(* PLC project Adressering.ecp, WAGO e!COCKPIT e!COCKPIT *)
(* stored: creationDateTime 2021-01-18T14:20:23.2110188, modificationDateTime 2021-01-18T11:51:27.6823754 *)

TYPE typVAV : STRUCT
  xReady : BOOL;  (* Status adr. *)
  xEnable : BOOL;  (* Enable MP blokk *)
  xAddress : BOOL;  (* Adresserer VAV *)
  xFailed : BOOL;  (* Tilbakemelding adressering (True = SerieNr inn og ut ikke stemmer) *)
  sSetStatus : STRING;  (* Status tilbakemelding naar adresseringen er i SET step *)
  sGetStatus : STRING;  (* Status tilbakemelding naar adresseringen er i GET step *)
  iSerialNr : typSerialNo;  (* Serie NR *)
  bPort : BYTE;  (* VAV Port *)
  bAddress : BYTE;  (* VAV Address *)
  rAirVolume_SP : REAL;  (* Settpunkt 0-100% *)
  rOutPosition : REAL;  (* Vinkel *)
  rOutAirVolume_perc : REAL;  (* Luftmengde i prosent *)
  rOutAirVolume_m3h : REAL;  (* Luftmengde i m3h *)
  wSensorValue : WORD;
  rVmin : REAL;
  rVmax : REAL;  (* Max vinkel *)
  xControlRangeIncreased : BOOL;
  xMecanicalOverload : BOOL;
  xActuatorHunting : BOOL;
  xSensorError : BOOL;
  xManualOpen : BOOL;
  xManualClose : BOOL;
  vMin : REAL;  (* Min luftmengde SP / 0-100 *)
  vNorm : REAL;  (* Settpunkt ved bevegelse / 0-100 *)
  vMax : REAL;  (* Maks luftmengde SP / 0-100 *)
  vSize : REAL;  (* Max kubikk *)
  vSetpoint_m3h : REAL;  (* SP% *)
  xdontoptimize : BOOL;  (* Fjerner VAV fra Optimizer *)
END_STRUCT;
END_TYPE

{attribute 'qualified_only'}
VAR_GLOBAL  (* STLV80_360 *)
  STLV80_A_360_6D201_SQ401 : typVAV := (xEnable := TRUE, vMin := 700, vNorm := 1400, vMax := 1400, vSize := 1750, bPort := 1, bAddress := 1, iSerialNr := (wYearAndWeek := 02045, wDayAndNumber := 50010, bTypeID := 158, bTestStation := 140));  (* / *)
  STLV80_A_360_6D301_SQ501 : typVAV := (xEnable := TRUE, vMin := 3200, vNorm := 3200, vMax := 3200, vSize := 5655, bPort := 1, bAddress := 2, iSerialNr := (wYearAndWeek := 02040, wDayAndNumber := 40202, bTypeID := 158, bTestStation := 153));  (* / *)
  STLV80_A_360_6A201_SQ401 : typVAV := (xEnable := TRUE, vMin := 2025, vNorm := 4050, vMax := 4050, vSize := 5655, bPort := 1, bAddress := 3, iSerialNr := (wYearAndWeek := 02040, wDayAndNumber := 40197, bTypeID := 158, bTestStation := 140));  (* / *)
  STLV80_A_360_6A201_SQ501 : typVAV := (xEnable := TRUE, vMin := 2700, vNorm := 2700, vMax := 2700, vSize := 5655, bPort := 1, bAddress := 4, iSerialNr := (wYearAndWeek := 02040, wDayAndNumber := 40201, bTypeID := 158, bTestStation := 159));  (* / *)
  STLV80_A_360_6C206_SQ501 : typVAV := (xEnable := TRUE, vMin := 300, vNorm := 300, vMax := 300, vSize := 700, bPort := 1, bAddress := 5, iSerialNr := (wYearAndWeek := 02105, wDayAndNumber := 10009, bTypeID := 158, bTestStation := 142));  (* / *)
  STLV80_A_360_6C206_SQ401 : typVAV := (xEnable := TRUE, vMin := 375, vNorm := 750, vMax := 750, vSize := 1750, bPort := 1, bAddress := 6, iSerialNr := (wYearAndWeek := 02045, wDayAndNumber := 50010, bTypeID := 158, bTestStation := 153));  (* / *)
  STLV80_A_360_7C201_SQ401 : typVAV := (xEnable := TRUE, vMin := 200, vNorm := 200, vMax := 200, vSize := 434, bPort := 1, bAddress := 7, iSerialNr := (wYearAndWeek := 02032, wDayAndNumber := 40145, bTypeID := 158, bTestStation := 158));  (* / *)
  STLV80_A_360_7C201_SQ501 : typVAV := (xEnable := TRUE, vMin := 400, vNorm := 400, vMax := 400, vSize := 700, bPort := 1, bAddress := 8, iSerialNr := (wYearAndWeek := 02042, wDayAndNumber := 10210, bTypeID := 158, bTestStation := 153));  (* / *)
  STLV80_A_360_6G201_SQ401 : typVAV := (xEnable := TRUE, vMin := 700, vNorm := 1400, vMax := 1400, vSize := 3619, bPort := 2, bAddress := 1, iSerialNr := (wYearAndWeek := 02042, wDayAndNumber := 10209, bTypeID := 158, bTestStation := 153));  (* / *)
  STLV80_A_360_6M201_SQ503 : typVAV := (xEnable := TRUE, vMin := 850, vNorm := 850, vMax := 850, vSize := 1060, bPort := 2, bAddress := 2, iSerialNr := (wYearAndWeek := 02005, wDayAndNumber := 20125, bTypeID := 158, bTestStation := 140));  (* / *)
  STLV80_A_360_6M201_SQ403 : typVAV := (xEnable := TRUE, vMin := 1225, vNorm := 2450, vMax := 2450, vSize := 5344, bPort := 2, bAddress := 3, iSerialNr := (wYearAndWeek := 02045, wDayAndNumber := 20003, bTypeID := 158, bTestStation := 140));  (* / *)
  STLV80_A_360_6M201_SQ402 : typVAV := (xEnable := TRUE, vMin := 700, vNorm := 1400, vMax := 1400, vSize := 4524, bPort := 2, bAddress := 4, iSerialNr := (wYearAndWeek := 02042, wDayAndNumber := 10207, bTypeID := 158, bTestStation := 153));  (* / *)
  STLV80_A_360_6M201_SQ502 : typVAV := (xEnable := TRUE, vMin := 3850, vNorm := 3850, vMax := 3850, vSize := 5655, bPort := 2, bAddress := 5, iSerialNr := (wYearAndWeek := 02040, wDayAndNumber := 40196, bTypeID := 158, bTestStation := 140));  (* / *)
  STLV80_A_360_6M201_SQ501 : typVAV := (xEnable := TRUE, vMin := 2600, vNorm := 2600, vMax := 2600, vSize := 5655, bPort := 2, bAddress := 6, iSerialNr := (wYearAndWeek := 02044, wDayAndNumber := 00121, bTypeID := 158, bTestStation := 164));  (* / *)
  STLV80_A_360_6M201_SQ401 : typVAV := (xEnable := TRUE, vMin := 900, vNorm := 1800, vMax := 1800, vSize := 5344, bPort := 2, bAddress := 7, iSerialNr := (wYearAndWeek := 02045, wDayAndNumber := 20006, bTypeID := 158, bTestStation := 140));  (* / *)
  STLV80_A_360_7O201_SQ401 : typVAV := (xEnable := TRUE, vMin := 200, vNorm := 200, vMax := 200, vSize := 700, bPort := 3, bAddress := 1, iSerialNr := (wYearAndWeek := 02032, wDayAndNumber := 40155, bTypeID := 158, bTestStation := 129));  (* / *)
  STLV80_A_360_7O201_SQ501 : typVAV := (xEnable := TRUE, vMin := 400, vNorm := 400, vMax := 400, vSize := 700, bPort := 3, bAddress := 2, iSerialNr := (wYearAndWeek := 02049, wDayAndNumber := 40093, bTypeID := 158, bTestStation := 142));  (* / *)
END_VAR

FUNCTION_BLOCK fbAutAd
  VAR_INPUT
    iSerialNr : typSerialNo;
    bPort : BYTE;
    bAddress : BYTE;
    xReset : BOOL;
    xNext : BOOL;
  END_VAR
  VAR_OUTPUT
    i : INT := 0;
    xFailed : BOOL;
    sSetStatus : STRING;
    sGetStatus : STRING;
  END_VAR
  VAR
    xLearn : BOOL;
    xRetry : BOOL;
    VAV_Addressing : fbMpBusAddressing;
  END_VAR

	//Resetter forgje VAVs verdier
	IF xReset THEN
		i:= 0;
		xRetry:= FALSE;
		xFailed:= FALSE;
		sSetStatus:= '';
		sGetStatus:= '';

//Begynner paa neste VAV
	ELSIF i<1 AND xNext THEN
		VAV_Addressing
		(
			bPortMpBus:= bPort,
			bAddress:= bAddress,
			typINSerialNo:= iSerialNr,
			xLearn:= xLearn
		);
		i:= 1;

//Skriver rett port og adresse til VAV naar blokken er klar
	ELSIF VAV_Addressing.xReady AND i=1 THEN
		VAV_Addressing
		(
			xSet:= TRUE,
			xLearn:= xLearn
		);
		i:= 2;

//Spoer etter serie nr som hoerer til port og adresse
	ELSIF VAV_Addressing.xReady AND i=2 THEN
		sSetStatus:= VAV_Addressing.sStatus;
		VAV_Addressing
		(
			xGetSerialNO:= TRUE,
			xLearn:= xLearn
		);
		i:= 3;

//Sjekker om serie nr. som tilhoerer port og adressen stemmer
	ELSIF VAV_Addressing.xReady AND i=3 THEN
		sGetStatus:= VAV_Addressing.sStatus;
		//Sjekker om serie nr stemmer
		IF xRetry AND VAV_Addressing.typOUTSerialNo.wYearAndWeek <> iSerialNr.wYearAndWeek OR VAV_Addressing.typOUTSerialNo.wDayAndNumber <> iSerialNr.wDayAndNumber OR VAV_Addressing.typOUTSerialNo.bTypeID <> iSerialNr.bTypeID OR VAV_Addressing.typOUTSerialNo.bTestStation <> iSerialNr.bTestStation THEN
			xRetry:= FALSE;
			xFailed:= TRUE;
			i:=4;
		ELSIF VAV_Addressing.typOUTSerialNo.wYearAndWeek <> iSerialNr.wYearAndWeek OR VAV_Addressing.typOUTSerialNo.wDayAndNumber <> iSerialNr.wDayAndNumber OR VAV_Addressing.typOUTSerialNo.bTypeID <> iSerialNr.bTypeID OR VAV_Addressing.typOUTSerialNo.bTestStation <> iSerialNr.bTestStation THEN
			xRetry:= TRUE;
			i:=1;
		ELSE
			i:=4;
		END_IF

//Resetter xSet og xGet, og Setter Port, adresse og serie nr. og henter status
	ELSE
		VAV_Addressing
		(
			bPortMpBus:= bPort,
			bAddress:= bAddress,
			typINSerialNo:= iSerialNr,
			xLearn:= xLearn,
			xSet:= FALSE,
			xGetSerialNO:= FALSE,
			xLearn:= xLearn
		);
	END_IF
				
END_FUNCTION_BLOCK

PROGRAM PRG_VAV_Adressering
  VAR
    xReset : BOOL;
    xRun : BOOL;
    xInit : BOOL := TRUE;
    Auto : fbAutAd;
    iLinje : INT;  (* Linje som skal adresseres *)
    iVAV : INT := 1;  (* VAV(adr.) som adresseres *)
  END_VAR

					IF xReset THEN
	Auto(xReset:= TRUE);
	xInit:= TRUE;
	xReset:= FALSE;
ELSIF xRun THEN

	IF STLV80_360.STLV80_A_360_6D201_SQ401.xAddress OR (iLinje = 1 AND iVAV = 1) THEN

		IF xInit THEN
			STLV80_360.STLV80_A_360_6D201_SQ401.xEnable:= FALSE;
			Auto(
				bPort:= STLV80_360.STLV80_A_360_6D201_SQ401.bPort,
				bAddress:= STLV80_360.STLV80_A_360_6D201_SQ401.bAddress,
				iSerialNr:= STLV80_360.STLV80_A_360_6D201_SQ401.iSerialNr,
				xNext:= TRUE,
				xReset:= FALSE
				);
			xInit:= FALSE;

		ELSIF Auto.i=4 THEN
			STLV80_360.STLV80_A_360_6D201_SQ401.sSetStatus:= Auto.sSetStatus;
				STLV80_360.STLV80_A_360_6D201_SQ401.sGetStatus:= Auto.sGetStatus;
				STLV80_360.STLV80_A_360_6D201_SQ401.xFailed:= Auto.xFailed;
				STLV80_360.STLV80_A_360_6D201_SQ401.xAddress:= FALSE;
				STLV80_360.STLV80_A_360_6D201_SQ401.xEnable:= TRUE;
				xReset:= TRUE;
				iVAV:=iVAV+1;

			ELSE
				Auto(xNext:= FALSE);
			END_IF

	ELSIF STLV80_360.STLV80_A_360_6D301_SQ501.xAddress OR (iLinje = 1 AND iVAV = 2) THEN

		IF xInit THEN
			STLV80_360.STLV80_A_360_6D301_SQ501.xEnable:= FALSE;
			Auto(
				bPort:= STLV80_360.STLV80_A_360_6D301_SQ501.bPort,
				bAddress:= STLV80_360.STLV80_A_360_6D301_SQ501.bAddress,
				iSerialNr:= STLV80_360.STLV80_A_360_6D301_SQ501.iSerialNr,
				xNext:= TRUE,
				xReset:= FALSE
				);
			xInit:= FALSE;

		ELSIF Auto.i=4 THEN
			STLV80_360.STLV80_A_360_6D301_SQ501.sSetStatus:= Auto.sSetStatus;
				STLV80_360.STLV80_A_360_6D301_SQ501.sGetStatus:= Auto.sGetStatus;
				STLV80_360.STLV80_A_360_6D301_SQ501.xFailed:= Auto.xFailed;
				STLV80_360.STLV80_A_360_6D301_SQ501.xAddress:= FALSE;
				STLV80_360.STLV80_A_360_6D301_SQ501.xEnable:= TRUE;
				xReset:= TRUE;
				iVAV:=iVAV+1;

			ELSE
				Auto(xNext:= FALSE);
			END_IF

	ELSIF STLV80_360.STLV80_A_360_6A201_SQ401.xAddress OR (iLinje = 1 AND iVAV = 3) THEN

		IF xInit THEN
			STLV80_360.STLV80_A_360_6A201_SQ401.xEnable:= FALSE;
			Auto(
				bPort:= STLV80_360.STLV80_A_360_6A201_SQ401.bPort,
				bAddress:= STLV80_360.STLV80_A_360_6A201_SQ401.bAddress,
				iSerialNr:= STLV80_360.STLV80_A_360_6A201_SQ401.iSerialNr,
				xNext:= TRUE,
				xReset:= FALSE
				);
			xInit:= FALSE;

		ELSIF Auto.i=4 THEN
			STLV80_360.STLV80_A_360_6A201_SQ401.sSetStatus:= Auto.sSetStatus;
				STLV80_360.STLV80_A_360_6A201_SQ401.sGetStatus:= Auto.sGetStatus;
				STLV80_360.STLV80_A_360_6A201_SQ401.xFailed:= Auto.xFailed;
				STLV80_360.STLV80_A_360_6A201_SQ401.xAddress:= FALSE;
				STLV80_360.STLV80_A_360_6A201_SQ401.xEnable:= TRUE;
				xReset:= TRUE;
				iVAV:=iVAV+1;

			ELSE
				Auto(xNext:= FALSE);
			END_IF

	ELSIF STLV80_360.STLV80_A_360_6A201_SQ501.xAddress OR (iLinje = 1 AND iVAV = 4) THEN

		IF xInit THEN
			STLV80_360.STLV80_A_360_6A201_SQ501.xEnable:= FALSE;
			Auto(
				bPort:= STLV80_360.STLV80_A_360_6A201_SQ501.bPort,
				bAddress:= STLV80_360.STLV80_A_360_6A201_SQ501.bAddress,
				iSerialNr:= STLV80_360.STLV80_A_360_6A201_SQ501.iSerialNr,
				xNext:= TRUE,
				xReset:= FALSE
				);
			xInit:= FALSE;

		ELSIF Auto.i=4 THEN
			STLV80_360.STLV80_A_360_6A201_SQ501.sSetStatus:= Auto.sSetStatus;
				STLV80_360.STLV80_A_360_6A201_SQ501.sGetStatus:= Auto.sGetStatus;
				STLV80_360.STLV80_A_360_6A201_SQ501.xFailed:= Auto.xFailed;
				STLV80_360.STLV80_A_360_6A201_SQ501.xAddress:= FALSE;
				STLV80_360.STLV80_A_360_6A201_SQ501.xEnable:= TRUE;
				xReset:= TRUE;
				iVAV:=iVAV+1;

			ELSE
				Auto(xNext:= FALSE);
			END_IF

	ELSIF STLV80_360.STLV80_A_360_6C206_SQ501.xAddress OR (iLinje = 1 AND iVAV = 5) THEN

		IF xInit THEN
			STLV80_360.STLV80_A_360_6C206_SQ501.xEnable:= FALSE;
			Auto(
				bPort:= STLV80_360.STLV80_A_360_6C206_SQ501.bPort,
				bAddress:= STLV80_360.STLV80_A_360_6C206_SQ501.bAddress,
				iSerialNr:= STLV80_360.STLV80_A_360_6C206_SQ501.iSerialNr,
				xNext:= TRUE,
				xReset:= FALSE
				);
			xInit:= FALSE;

		ELSIF Auto.i=4 THEN
			STLV80_360.STLV80_A_360_6C206_SQ501.sSetStatus:= Auto.sSetStatus;
				STLV80_360.STLV80_A_360_6C206_SQ501.sGetStatus:= Auto.sGetStatus;
				STLV80_360.STLV80_A_360_6C206_SQ501.xFailed:= Auto.xFailed;
				STLV80_360.STLV80_A_360_6C206_SQ501.xAddress:= FALSE;
				STLV80_360.STLV80_A_360_6C206_SQ501.xEnable:= TRUE;
				xReset:= TRUE;
				iVAV:=iVAV+1;

			ELSE
				Auto(xNext:= FALSE);
			END_IF

	ELSIF STLV80_360.STLV80_A_360_6C206_SQ401.xAddress OR (iLinje = 1 AND iVAV = 6) THEN

		IF xInit THEN
			STLV80_360.STLV80_A_360_6C206_SQ401.xEnable:= FALSE;
			Auto(
				bPort:= STLV80_360.STLV80_A_360_6C206_SQ401.bPort,
				bAddress:= STLV80_360.STLV80_A_360_6C206_SQ401.bAddress,
				iSerialNr:= STLV80_360.STLV80_A_360_6C206_SQ401.iSerialNr,
				xNext:= TRUE,
				xReset:= FALSE
				);
			xInit:= FALSE;

		ELSIF Auto.i=4 THEN
			STLV80_360.STLV80_A_360_6C206_SQ401.sSetStatus:= Auto.sSetStatus;
				STLV80_360.STLV80_A_360_6C206_SQ401.sGetStatus:= Auto.sGetStatus;
				STLV80_360.STLV80_A_360_6C206_SQ401.xFailed:= Auto.xFailed;
				STLV80_360.STLV80_A_360_6C206_SQ401.xAddress:= FALSE;
				STLV80_360.STLV80_A_360_6C206_SQ401.xEnable:= TRUE;
				xReset:= TRUE;
				iVAV:=iVAV+1;

			ELSE
				Auto(xNext:= FALSE);
			END_IF

	ELSIF STLV80_360.STLV80_A_360_7C201_SQ401.xAddress OR (iLinje = 1 AND iVAV = 7) THEN

		IF xInit THEN
			STLV80_360.STLV80_A_360_7C201_SQ401.xEnable:= FALSE;
			Auto(
				bPort:= STLV80_360.STLV80_A_360_7C201_SQ401.bPort,
				bAddress:= STLV80_360.STLV80_A_360_7C201_SQ401.bAddress,
				iSerialNr:= STLV80_360.STLV80_A_360_7C201_SQ401.iSerialNr,
				xNext:= TRUE,
				xReset:= FALSE
				);
			xInit:= FALSE;

		ELSIF Auto.i=4 THEN
			STLV80_360.STLV80_A_360_7C201_SQ401.sSetStatus:= Auto.sSetStatus;
				STLV80_360.STLV80_A_360_7C201_SQ401.sGetStatus:= Auto.sGetStatus;
				STLV80_360.STLV80_A_360_7C201_SQ401.xFailed:= Auto.xFailed;
				STLV80_360.STLV80_A_360_7C201_SQ401.xAddress:= FALSE;
				STLV80_360.STLV80_A_360_7C201_SQ401.xEnable:= TRUE;
				xReset:= TRUE;
				iVAV:=iVAV+1;

			ELSE
				Auto(xNext:= FALSE);
			END_IF

	ELSIF STLV80_360.STLV80_A_360_7C201_SQ501.xAddress OR (iLinje = 1 AND iVAV = 8) THEN

		IF xInit THEN
			STLV80_360.STLV80_A_360_7C201_SQ501.xEnable:= FALSE;
			Auto(
				bPort:= STLV80_360.STLV80_A_360_7C201_SQ501.bPort,
				bAddress:= STLV80_360.STLV80_A_360_7C201_SQ501.bAddress,
				iSerialNr:= STLV80_360.STLV80_A_360_7C201_SQ501.iSerialNr,
				xNext:= TRUE,
				xReset:= FALSE
				);
			xInit:= FALSE;

		ELSIF Auto.i=4 THEN
			STLV80_360.STLV80_A_360_7C201_SQ501.sSetStatus:= Auto.sSetStatus;
				STLV80_360.STLV80_A_360_7C201_SQ501.sGetStatus:= Auto.sGetStatus;
				STLV80_360.STLV80_A_360_7C201_SQ501.xFailed:= Auto.xFailed;
				STLV80_360.STLV80_A_360_7C201_SQ501.xAddress:= FALSE;
				STLV80_360.STLV80_A_360_7C201_SQ501.xEnable:= TRUE;
				xReset:= TRUE;
				iVAV:=iVAV+1;

			ELSE
				Auto(xNext:= FALSE);
			END_IF

	ELSIF STLV80_360.STLV80_A_360_6G201_SQ401.xAddress OR (iLinje = 2 AND iVAV = 1) THEN

		IF xInit THEN
			STLV80_360.STLV80_A_360_6G201_SQ401.xEnable:= FALSE;
			Auto(
				bPort:= STLV80_360.STLV80_A_360_6G201_SQ401.bPort,
				bAddress:= STLV80_360.STLV80_A_360_6G201_SQ401.bAddress,
				iSerialNr:= STLV80_360.STLV80_A_360_6G201_SQ401.iSerialNr,
				xNext:= TRUE,
				xReset:= FALSE
				);
			xInit:= FALSE;

		ELSIF Auto.i=4 THEN
			STLV80_360.STLV80_A_360_6G201_SQ401.sSetStatus:= Auto.sSetStatus;
				STLV80_360.STLV80_A_360_6G201_SQ401.sGetStatus:= Auto.sGetStatus;
				STLV80_360.STLV80_A_360_6G201_SQ401.xFailed:= Auto.xFailed;
				STLV80_360.STLV80_A_360_6G201_SQ401.xAddress:= FALSE;
				STLV80_360.STLV80_A_360_6G201_SQ401.xEnable:= TRUE;
				xReset:= TRUE;
				iVAV:=iVAV+1;

			ELSE
				Auto(xNext:= FALSE);
			END_IF

	ELSIF STLV80_360.STLV80_A_360_6M201_SQ503.xAddress OR (iLinje = 2 AND iVAV = 2) THEN

		IF xInit THEN
			STLV80_360.STLV80_A_360_6M201_SQ503.xEnable:= FALSE;
			Auto(
				bPort:= STLV80_360.STLV80_A_360_6M201_SQ503.bPort,
				bAddress:= STLV80_360.STLV80_A_360_6M201_SQ503.bAddress,
				iSerialNr:= STLV80_360.STLV80_A_360_6M201_SQ503.iSerialNr,
				xNext:= TRUE,
				xReset:= FALSE
				);
			xInit:= FALSE;

		ELSIF Auto.i=4 THEN
			STLV80_360.STLV80_A_360_6M201_SQ503.sSetStatus:= Auto.sSetStatus;
				STLV80_360.STLV80_A_360_6M201_SQ503.sGetStatus:= Auto.sGetStatus;
				STLV80_360.STLV80_A_360_6M201_SQ503.xFailed:= Auto.xFailed;
				STLV80_360.STLV80_A_360_6M201_SQ503.xAddress:= FALSE;
				STLV80_360.STLV80_A_360_6M201_SQ503.xEnable:= TRUE;
				xReset:= TRUE;
				iVAV:=iVAV+1;

			ELSE
				Auto(xNext:= FALSE);
			END_IF

	ELSIF STLV80_360.STLV80_A_360_6M201_SQ403.xAddress OR (iLinje = 2 AND iVAV = 3) THEN

		IF xInit THEN
			STLV80_360.STLV80_A_360_6M201_SQ403.xEnable:= FALSE;
			Auto(
				bPort:= STLV80_360.STLV80_A_360_6M201_SQ403.bPort,
				bAddress:= STLV80_360.STLV80_A_360_6M201_SQ403.bAddress,
				iSerialNr:= STLV80_360.STLV80_A_360_6M201_SQ403.iSerialNr,
				xNext:= TRUE,
				xReset:= FALSE
				);
			xInit:= FALSE;

		ELSIF Auto.i=4 THEN
			STLV80_360.STLV80_A_360_6M201_SQ403.sSetStatus:= Auto.sSetStatus;
				STLV80_360.STLV80_A_360_6M201_SQ403.sGetStatus:= Auto.sGetStatus;
				STLV80_360.STLV80_A_360_6M201_SQ403.xFailed:= Auto.xFailed;
				STLV80_360.STLV80_A_360_6M201_SQ403.xAddress:= FALSE;
				STLV80_360.STLV80_A_360_6M201_SQ403.xEnable:= TRUE;
				xReset:= TRUE;
				iVAV:=iVAV+1;

			ELSE
				Auto(xNext:= FALSE);
			END_IF

	ELSIF STLV80_360.STLV80_A_360_6M201_SQ402.xAddress OR (iLinje = 2 AND iVAV = 4) THEN

		IF xInit THEN
			STLV80_360.STLV80_A_360_6M201_SQ402.xEnable:= FALSE;
			Auto(
				bPort:= STLV80_360.STLV80_A_360_6M201_SQ402.bPort,
				bAddress:= STLV80_360.STLV80_A_360_6M201_SQ402.bAddress,
				iSerialNr:= STLV80_360.STLV80_A_360_6M201_SQ402.iSerialNr,
				xNext:= TRUE,
				xReset:= FALSE
				);
			xInit:= FALSE;

		ELSIF Auto.i=4 THEN
			STLV80_360.STLV80_A_360_6M201_SQ402.sSetStatus:= Auto.sSetStatus;
				STLV80_360.STLV80_A_360_6M201_SQ402.sGetStatus:= Auto.sGetStatus;
				STLV80_360.STLV80_A_360_6M201_SQ402.xFailed:= Auto.xFailed;
				STLV80_360.STLV80_A_360_6M201_SQ402.xAddress:= FALSE;
				STLV80_360.STLV80_A_360_6M201_SQ402.xEnable:= TRUE;
				xReset:= TRUE;
				iVAV:=iVAV+1;

			ELSE
				Auto(xNext:= FALSE);
			END_IF

	ELSIF STLV80_360.STLV80_A_360_6M201_SQ502.xAddress OR (iLinje = 2 AND iVAV = 5) THEN

		IF xInit THEN
			STLV80_360.STLV80_A_360_6M201_SQ502.xEnable:= FALSE;
			Auto(
				bPort:= STLV80_360.STLV80_A_360_6M201_SQ502.bPort,
				bAddress:= STLV80_360.STLV80_A_360_6M201_SQ502.bAddress,
				iSerialNr:= STLV80_360.STLV80_A_360_6M201_SQ502.iSerialNr,
				xNext:= TRUE,
				xReset:= FALSE
				);
			xInit:= FALSE;

		ELSIF Auto.i=4 THEN
			STLV80_360.STLV80_A_360_6M201_SQ502.sSetStatus:= Auto.sSetStatus;
				STLV80_360.STLV80_A_360_6M201_SQ502.sGetStatus:= Auto.sGetStatus;
				STLV80_360.STLV80_A_360_6M201_SQ502.xFailed:= Auto.xFailed;
				STLV80_360.STLV80_A_360_6M201_SQ502.xAddress:= FALSE;
				STLV80_360.STLV80_A_360_6M201_SQ502.xEnable:= TRUE;
				xReset:= TRUE;
				iVAV:=iVAV+1;

			ELSE
				Auto(xNext:= FALSE);
			END_IF

	ELSIF STLV80_360.STLV80_A_360_6M201_SQ501.xAddress OR (iLinje = 2 AND iVAV = 6) THEN

		IF xInit THEN
			STLV80_360.STLV80_A_360_6M201_SQ501.xEnable:= FALSE;
			Auto(
				bPort:= STLV80_360.STLV80_A_360_6M201_SQ501.bPort,
				bAddress:= STLV80_360.STLV80_A_360_6M201_SQ501.bAddress,
				iSerialNr:= STLV80_360.STLV80_A_360_6M201_SQ501.iSerialNr,
				xNext:= TRUE,
				xReset:= FALSE
				);
			xInit:= FALSE;

		ELSIF Auto.i=4 THEN
			STLV80_360.STLV80_A_360_6M201_SQ501.sSetStatus:= Auto.sSetStatus;
				STLV80_360.STLV80_A_360_6M201_SQ501.sGetStatus:= Auto.sGetStatus;
				STLV80_360.STLV80_A_360_6M201_SQ501.xFailed:= Auto.xFailed;
				STLV80_360.STLV80_A_360_6M201_SQ501.xAddress:= FALSE;
				STLV80_360.STLV80_A_360_6M201_SQ501.xEnable:= TRUE;
				xReset:= TRUE;
				iVAV:=iVAV+1;

			ELSE
				Auto(xNext:= FALSE);
			END_IF

	ELSIF STLV80_360.STLV80_A_360_6M201_SQ401.xAddress OR (iLinje = 2 AND iVAV = 7) THEN

		IF xInit THEN
			STLV80_360.STLV80_A_360_6M201_SQ401.xEnable:= FALSE;
			Auto(
				bPort:= STLV80_360.STLV80_A_360_6M201_SQ401.bPort,
				bAddress:= STLV80_360.STLV80_A_360_6M201_SQ401.bAddress,
				iSerialNr:= STLV80_360.STLV80_A_360_6M201_SQ401.iSerialNr,
				xNext:= TRUE,
				xReset:= FALSE
				);
			xInit:= FALSE;

		ELSIF Auto.i=4 THEN
			STLV80_360.STLV80_A_360_6M201_SQ401.sSetStatus:= Auto.sSetStatus;
				STLV80_360.STLV80_A_360_6M201_SQ401.sGetStatus:= Auto.sGetStatus;
				STLV80_360.STLV80_A_360_6M201_SQ401.xFailed:= Auto.xFailed;
				STLV80_360.STLV80_A_360_6M201_SQ401.xAddress:= FALSE;
				STLV80_360.STLV80_A_360_6M201_SQ401.xEnable:= TRUE;
				xReset:= TRUE;
				iVAV:=iVAV+1;

			ELSE
				Auto(xNext:= FALSE);
			END_IF

	ELSIF STLV80_360.STLV80_A_360_7O201_SQ401.xAddress OR (iLinje = 3 AND iVAV = 1) THEN

		IF xInit THEN
			STLV80_360.STLV80_A_360_7O201_SQ401.xEnable:= FALSE;
			Auto(
				bPort:= STLV80_360.STLV80_A_360_7O201_SQ401.bPort,
				bAddress:= STLV80_360.STLV80_A_360_7O201_SQ401.bAddress,
				iSerialNr:= STLV80_360.STLV80_A_360_7O201_SQ401.iSerialNr,
				xNext:= TRUE,
				xReset:= FALSE
				);
			xInit:= FALSE;

		ELSIF Auto.i=4 THEN
			STLV80_360.STLV80_A_360_7O201_SQ401.sSetStatus:= Auto.sSetStatus;
				STLV80_360.STLV80_A_360_7O201_SQ401.sGetStatus:= Auto.sGetStatus;
				STLV80_360.STLV80_A_360_7O201_SQ401.xFailed:= Auto.xFailed;
				STLV80_360.STLV80_A_360_7O201_SQ401.xAddress:= FALSE;
				STLV80_360.STLV80_A_360_7O201_SQ401.xEnable:= TRUE;
				xReset:= TRUE;
				iVAV:=iVAV+1;

			ELSE
				Auto(xNext:= FALSE);
			END_IF

	ELSIF STLV80_360.STLV80_A_360_7O201_SQ501.xAddress OR (iLinje = 3 AND iVAV = 2) THEN

		IF xInit THEN
			STLV80_360.STLV80_A_360_7O201_SQ501.xEnable:= FALSE;
			Auto(
				bPort:= STLV80_360.STLV80_A_360_7O201_SQ501.bPort,
				bAddress:= STLV80_360.STLV80_A_360_7O201_SQ501.bAddress,
				iSerialNr:= STLV80_360.STLV80_A_360_7O201_SQ501.iSerialNr,
				xNext:= TRUE,
				xReset:= FALSE
				);
			xInit:= FALSE;

		ELSIF Auto.i=4 THEN
			STLV80_360.STLV80_A_360_7O201_SQ501.sSetStatus:= Auto.sSetStatus;
				STLV80_360.STLV80_A_360_7O201_SQ501.sGetStatus:= Auto.sGetStatus;
				STLV80_360.STLV80_A_360_7O201_SQ501.xFailed:= Auto.xFailed;
				STLV80_360.STLV80_A_360_7O201_SQ501.xAddress:= FALSE;
				STLV80_360.STLV80_A_360_7O201_SQ501.xEnable:= TRUE;
				xReset:= TRUE;
				iVAV:=iVAV+1;

			ELSE
				Auto(xNext:= FALSE);
			END_IF

	ELSIF iVAV > 8 THEN
			iVAV:= 0;
		ELSIF iVAV > 0  THEN
			iVAV:= (iVAV+1);
		END_IF
END_IF

				
END_PROGRAM

PROGRAM PRG_MP1
  VAR
    xSet : BOOL;  (* Felles *)
    xRead : BOOL;
    FbMpbusMaster_1 : FbMpbusMaster;  (* Master *)
    oStatus_M1 : WagoSysErrorBase.FbResult;
    sStatus_M1 : STRING;
    FbMpbus_1 : FbMpBusVav;  (* Linje 1. Adresse 1. VAV STLV80_A_360_6D201_SQ401 *)
    oStatus_1 : WagoSysErrorBase.FbResult;
    sStatus_1 : STRING;
    FbMpbus_2 : FbMpBusVav;  (* Linje 1. Adresse 2. VAV STLV80_A_360_6D301_SQ501 *)
    oStatus_2 : WagoSysErrorBase.FbResult;
    sStatus_2 : STRING;
    FbMpbus_3 : FbMpBusVav;  (* Linje 1. Adresse 3. VAV STLV80_A_360_6A201_SQ401 *)
    oStatus_3 : WagoSysErrorBase.FbResult;
    sStatus_3 : STRING;
    FbMpbus_4 : FbMpBusVav;  (* Linje 1. Adresse 4. VAV STLV80_A_360_6A201_SQ501 *)
    oStatus_4 : WagoSysErrorBase.FbResult;
    sStatus_4 : STRING;
    FbMpbus_5 : FbMpBusVav;  (* Linje 1. Adresse 5. VAV STLV80_A_360_6C206_SQ501 *)
    oStatus_5 : WagoSysErrorBase.FbResult;
    sStatus_5 : STRING;
    FbMpbus_6 : FbMpBusVav;  (* Linje 1. Adresse 6. VAV STLV80_A_360_6C206_SQ401 *)
    oStatus_6 : WagoSysErrorBase.FbResult;
    sStatus_6 : STRING;
    FbMpbus_7 : FbMpBusVav;  (* Linje 1. Adresse 7. VAV STLV80_A_360_7C201_SQ401 *)
    oStatus_7 : WagoSysErrorBase.FbResult;
    sStatus_7 : STRING;
    FbMpbus_8 : FbMpBusVav;  (* Linje 1. Adresse 8. VAV STLV80_A_360_7C201_SQ501 *)
    oStatus_8 : WagoSysErrorBase.FbResult;
    sStatus_8 : STRING;
  END_VAR

(* CFC diagram, written out as Structured Text *)
FbMpbusMaster_1(I_Port := IoConfig_Globals.MP_Bus_Master, bPortMpBus := 1);
oStatus_M1 := FbMpbusMaster_1.oStatus;
sStatus_M1 := FbMpbusMaster_1.sStatus;
(* STLV80_A_360_6D201_SQ401 *)
FbMpbus_1(xEnable := STLV80_360.STLV80_A_360_6D201_SQ401.xEnable, bPortMpBus := 1, bAddress := 1, tCycleTime := t#500ms, rAirVolume := STLV80_360.STLV80_A_360_6D201_SQ401.rAirVolume_SP, rMinAirVolume := 0, rMaxAirVolume := 100, xSet := xSet, xRead := xRead, bSensorType := 0, xManualOpen := STLV80_360.STLV80_A_360_6D201_SQ401.xManualOpen, xManualClose := STLV80_360.STLV80_A_360_6D201_SQ401.xManualClose);
oStatus_1 := FbMpbus_1.oStatus;
sStatus_1 := FbMpbus_1.sStatus;
STLV80_360.STLV80_A_360_6D201_SQ401.xReady := FbMpbus_1.xReady;
STLV80_360.STLV80_A_360_6D201_SQ401.rOutPosition := FbMpbus_1.rOutPosition;
STLV80_360.STLV80_A_360_6D201_SQ401.rOutAirVolume_perc := FbMpbus_1.rOutAirVolume_perc;
STLV80_360.STLV80_A_360_6D201_SQ401.rOutAirVolume_m3h := FbMpbus_1.rOutAirVolume_m3_h;
STLV80_360.STLV80_A_360_6D201_SQ401.wSensorValue := FbMpbus_1.wSensorValue;
STLV80_360.STLV80_A_360_6D201_SQ401.rVmin := FbMpbus_1.rVmin;
STLV80_360.STLV80_A_360_6D201_SQ401.rVmax := FbMpbus_1.rVmax;
STLV80_360.STLV80_A_360_6D201_SQ401.xControlRangeIncreased := FbMpbus_1.xControlRangeIncreased;
STLV80_360.STLV80_A_360_6D201_SQ401.xMecanicalOverload := FbMpbus_1.xMecanicalOverload;
STLV80_360.STLV80_A_360_6D201_SQ401.xActuatorHunting := FbMpbus_1.xActuatorHunting;
STLV80_360.STLV80_A_360_6D201_SQ401.xSensorError := FbMpbus_1.xSensorError;
(* STLV80_A_360_6D301_SQ501 *)
FbMpbus_2(xEnable := STLV80_360.STLV80_A_360_6D301_SQ501.xEnable, bPortMpBus := 1, bAddress := 2, tCycleTime := t#500ms, rAirVolume := STLV80_360.STLV80_A_360_6D301_SQ501.rAirVolume_SP, rMinAirVolume := 0, rMaxAirVolume := 100, xSet := xSet, xRead := xRead, bSensorType := 0, xManualOpen := STLV80_360.STLV80_A_360_6D301_SQ501.xManualOpen, xManualClose := STLV80_360.STLV80_A_360_6D301_SQ501.xManualClose);
oStatus_2 := FbMpbus_2.oStatus;
sStatus_2 := FbMpbus_2.sStatus;
STLV80_360.STLV80_A_360_6D301_SQ501.xReady := FbMpbus_2.xReady;
STLV80_360.STLV80_A_360_6D301_SQ501.rOutPosition := FbMpbus_2.rOutPosition;
STLV80_360.STLV80_A_360_6D301_SQ501.rOutAirVolume_perc := FbMpbus_2.rOutAirVolume_perc;
STLV80_360.STLV80_A_360_6D301_SQ501.rOutAirVolume_m3h := FbMpbus_2.rOutAirVolume_m3_h;
STLV80_360.STLV80_A_360_6D301_SQ501.wSensorValue := FbMpbus_2.wSensorValue;
STLV80_360.STLV80_A_360_6D301_SQ501.rVmin := FbMpbus_2.rVmin;
STLV80_360.STLV80_A_360_6D301_SQ501.rVmax := FbMpbus_2.rVmax;
STLV80_360.STLV80_A_360_6D301_SQ501.xControlRangeIncreased := FbMpbus_2.xControlRangeIncreased;
STLV80_360.STLV80_A_360_6D301_SQ501.xMecanicalOverload := FbMpbus_2.xMecanicalOverload;
STLV80_360.STLV80_A_360_6D301_SQ501.xActuatorHunting := FbMpbus_2.xActuatorHunting;
STLV80_360.STLV80_A_360_6D301_SQ501.xSensorError := FbMpbus_2.xSensorError;
(* STLV80_A_360_6A201_SQ401 *)
FbMpbus_3(xEnable := STLV80_360.STLV80_A_360_6A201_SQ401.xEnable, bPortMpBus := 1, bAddress := 3, tCycleTime := t#500ms, rAirVolume := STLV80_360.STLV80_A_360_6A201_SQ401.rAirVolume_SP, rMinAirVolume := 0, rMaxAirVolume := 100, xSet := xSet, xRead := xRead, bSensorType := 0, xManualOpen := STLV80_360.STLV80_A_360_6A201_SQ401.xManualOpen, xManualClose := STLV80_360.STLV80_A_360_6A201_SQ401.xManualClose);
oStatus_3 := FbMpbus_3.oStatus;
sStatus_3 := FbMpbus_3.sStatus;
STLV80_360.STLV80_A_360_6A201_SQ401.xReady := FbMpbus_3.xReady;
STLV80_360.STLV80_A_360_6A201_SQ401.rOutPosition := FbMpbus_3.rOutPosition;
STLV80_360.STLV80_A_360_6A201_SQ401.rOutAirVolume_perc := FbMpbus_3.rOutAirVolume_perc;
STLV80_360.STLV80_A_360_6A201_SQ401.rOutAirVolume_m3h := FbMpbus_3.rOutAirVolume_m3_h;
STLV80_360.STLV80_A_360_6A201_SQ401.wSensorValue := FbMpbus_3.wSensorValue;
STLV80_360.STLV80_A_360_6A201_SQ401.rVmin := FbMpbus_3.rVmin;
STLV80_360.STLV80_A_360_6A201_SQ401.rVmax := FbMpbus_3.rVmax;
STLV80_360.STLV80_A_360_6A201_SQ401.xControlRangeIncreased := FbMpbus_3.xControlRangeIncreased;
STLV80_360.STLV80_A_360_6A201_SQ401.xMecanicalOverload := FbMpbus_3.xMecanicalOverload;
STLV80_360.STLV80_A_360_6A201_SQ401.xActuatorHunting := FbMpbus_3.xActuatorHunting;
STLV80_360.STLV80_A_360_6A201_SQ401.xSensorError := FbMpbus_3.xSensorError;
(* STLV80_A_360_6A201_SQ501 *)
FbMpbus_4(xEnable := STLV80_360.STLV80_A_360_6A201_SQ501.xEnable, bPortMpBus := 1, bAddress := 4, tCycleTime := t#500ms, rAirVolume := STLV80_360.STLV80_A_360_6A201_SQ501.rAirVolume_SP, rMinAirVolume := 0, rMaxAirVolume := 100, xSet := xSet, xRead := xRead, bSensorType := 0, xManualOpen := STLV80_360.STLV80_A_360_6A201_SQ501.xManualOpen, xManualClose := STLV80_360.STLV80_A_360_6A201_SQ501.xManualClose);
oStatus_4 := FbMpbus_4.oStatus;
sStatus_4 := FbMpbus_4.sStatus;
STLV80_360.STLV80_A_360_6A201_SQ501.xReady := FbMpbus_4.xReady;
STLV80_360.STLV80_A_360_6A201_SQ501.rOutPosition := FbMpbus_4.rOutPosition;
STLV80_360.STLV80_A_360_6A201_SQ501.rOutAirVolume_perc := FbMpbus_4.rOutAirVolume_perc;
STLV80_360.STLV80_A_360_6A201_SQ501.rOutAirVolume_m3h := FbMpbus_4.rOutAirVolume_m3_h;
STLV80_360.STLV80_A_360_6A201_SQ501.wSensorValue := FbMpbus_4.wSensorValue;
STLV80_360.STLV80_A_360_6A201_SQ501.rVmin := FbMpbus_4.rVmin;
STLV80_360.STLV80_A_360_6A201_SQ501.rVmax := FbMpbus_4.rVmax;
STLV80_360.STLV80_A_360_6A201_SQ501.xControlRangeIncreased := FbMpbus_4.xControlRangeIncreased;
STLV80_360.STLV80_A_360_6A201_SQ501.xMecanicalOverload := FbMpbus_4.xMecanicalOverload;
STLV80_360.STLV80_A_360_6A201_SQ501.xActuatorHunting := FbMpbus_4.xActuatorHunting;
STLV80_360.STLV80_A_360_6A201_SQ501.xSensorError := FbMpbus_4.xSensorError;
(* STLV80_A_360_6C206_SQ501 *)
FbMpbus_5(xEnable := STLV80_360.STLV80_A_360_6C206_SQ501.xEnable, bPortMpBus := 1, bAddress := 5, tCycleTime := t#500ms, rAirVolume := STLV80_360.STLV80_A_360_6C206_SQ501.rAirVolume_SP, rMinAirVolume := 0, rMaxAirVolume := 100, xSet := xSet, xRead := xRead, bSensorType := 0, xManualOpen := STLV80_360.STLV80_A_360_6C206_SQ501.xManualOpen, xManualClose := STLV80_360.STLV80_A_360_6C206_SQ501.xManualClose);
oStatus_5 := FbMpbus_5.oStatus;
sStatus_5 := FbMpbus_5.sStatus;
STLV80_360.STLV80_A_360_6C206_SQ501.xReady := FbMpbus_5.xReady;
STLV80_360.STLV80_A_360_6C206_SQ501.rOutPosition := FbMpbus_5.rOutPosition;
STLV80_360.STLV80_A_360_6C206_SQ501.rOutAirVolume_perc := FbMpbus_5.rOutAirVolume_perc;
STLV80_360.STLV80_A_360_6C206_SQ501.rOutAirVolume_m3h := FbMpbus_5.rOutAirVolume_m3_h;
STLV80_360.STLV80_A_360_6C206_SQ501.wSensorValue := FbMpbus_5.wSensorValue;
STLV80_360.STLV80_A_360_6C206_SQ501.rVmin := FbMpbus_5.rVmin;
STLV80_360.STLV80_A_360_6C206_SQ501.rVmax := FbMpbus_5.rVmax;
STLV80_360.STLV80_A_360_6C206_SQ501.xControlRangeIncreased := FbMpbus_5.xControlRangeIncreased;
STLV80_360.STLV80_A_360_6C206_SQ501.xMecanicalOverload := FbMpbus_5.xMecanicalOverload;
STLV80_360.STLV80_A_360_6C206_SQ501.xActuatorHunting := FbMpbus_5.xActuatorHunting;
STLV80_360.STLV80_A_360_6C206_SQ501.xSensorError := FbMpbus_5.xSensorError;
(* STLV80_A_360_6C206_SQ401 *)
FbMpbus_6(xEnable := STLV80_360.STLV80_A_360_6C206_SQ401.xEnable, bPortMpBus := 1, bAddress := 6, tCycleTime := t#500ms, rAirVolume := STLV80_360.STLV80_A_360_6C206_SQ401.rAirVolume_SP, rMinAirVolume := 0, rMaxAirVolume := 100, xSet := xSet, xRead := xRead, bSensorType := 0, xManualOpen := STLV80_360.STLV80_A_360_6C206_SQ401.xManualOpen, xManualClose := STLV80_360.STLV80_A_360_6C206_SQ401.xManualClose);
oStatus_6 := FbMpbus_6.oStatus;
sStatus_6 := FbMpbus_6.sStatus;
STLV80_360.STLV80_A_360_6C206_SQ401.xReady := FbMpbus_6.xReady;
STLV80_360.STLV80_A_360_6C206_SQ401.rOutPosition := FbMpbus_6.rOutPosition;
STLV80_360.STLV80_A_360_6C206_SQ401.rOutAirVolume_perc := FbMpbus_6.rOutAirVolume_perc;
STLV80_360.STLV80_A_360_6C206_SQ401.rOutAirVolume_m3h := FbMpbus_6.rOutAirVolume_m3_h;
STLV80_360.STLV80_A_360_6C206_SQ401.wSensorValue := FbMpbus_6.wSensorValue;
STLV80_360.STLV80_A_360_6C206_SQ401.rVmin := FbMpbus_6.rVmin;
STLV80_360.STLV80_A_360_6C206_SQ401.rVmax := FbMpbus_6.rVmax;
STLV80_360.STLV80_A_360_6C206_SQ401.xControlRangeIncreased := FbMpbus_6.xControlRangeIncreased;
STLV80_360.STLV80_A_360_6C206_SQ401.xMecanicalOverload := FbMpbus_6.xMecanicalOverload;
STLV80_360.STLV80_A_360_6C206_SQ401.xActuatorHunting := FbMpbus_6.xActuatorHunting;
STLV80_360.STLV80_A_360_6C206_SQ401.xSensorError := FbMpbus_6.xSensorError;
(* STLV80_A_360_7C201_SQ401 *)
FbMpbus_7(xEnable := STLV80_360.STLV80_A_360_7C201_SQ401.xEnable, bPortMpBus := 1, bAddress := 7, tCycleTime := t#500ms, rAirVolume := STLV80_360.STLV80_A_360_7C201_SQ401.rAirVolume_SP, rMinAirVolume := 0, rMaxAirVolume := 100, xSet := xSet, xRead := xRead, bSensorType := 0, xManualOpen := STLV80_360.STLV80_A_360_7C201_SQ401.xManualOpen, xManualClose := STLV80_360.STLV80_A_360_7C201_SQ401.xManualClose);
oStatus_7 := FbMpbus_7.oStatus;
sStatus_7 := FbMpbus_7.sStatus;
STLV80_360.STLV80_A_360_7C201_SQ401.xReady := FbMpbus_7.xReady;
STLV80_360.STLV80_A_360_7C201_SQ401.rOutPosition := FbMpbus_7.rOutPosition;
STLV80_360.STLV80_A_360_7C201_SQ401.rOutAirVolume_perc := FbMpbus_7.rOutAirVolume_perc;
STLV80_360.STLV80_A_360_7C201_SQ401.rOutAirVolume_m3h := FbMpbus_7.rOutAirVolume_m3_h;
STLV80_360.STLV80_A_360_7C201_SQ401.wSensorValue := FbMpbus_7.wSensorValue;
STLV80_360.STLV80_A_360_7C201_SQ401.rVmin := FbMpbus_7.rVmin;
STLV80_360.STLV80_A_360_7C201_SQ401.rVmax := FbMpbus_7.rVmax;
STLV80_360.STLV80_A_360_7C201_SQ401.xControlRangeIncreased := FbMpbus_7.xControlRangeIncreased;
STLV80_360.STLV80_A_360_7C201_SQ401.xMecanicalOverload := FbMpbus_7.xMecanicalOverload;
STLV80_360.STLV80_A_360_7C201_SQ401.xActuatorHunting := FbMpbus_7.xActuatorHunting;
STLV80_360.STLV80_A_360_7C201_SQ401.xSensorError := FbMpbus_7.xSensorError;
(* STLV80_A_360_7C201_SQ501 *)
FbMpbus_8(xEnable := STLV80_360.STLV80_A_360_7C201_SQ501.xEnable, bPortMpBus := 1, bAddress := 8, tCycleTime := t#500ms, rAirVolume := STLV80_360.STLV80_A_360_7C201_SQ501.rAirVolume_SP, rMinAirVolume := 0, rMaxAirVolume := 100, xSet := xSet, xRead := xRead, bSensorType := 0, xManualOpen := STLV80_360.STLV80_A_360_7C201_SQ501.xManualOpen, xManualClose := STLV80_360.STLV80_A_360_7C201_SQ501.xManualClose);
oStatus_8 := FbMpbus_8.oStatus;
sStatus_8 := FbMpbus_8.sStatus;
STLV80_360.STLV80_A_360_7C201_SQ501.xReady := FbMpbus_8.xReady;
STLV80_360.STLV80_A_360_7C201_SQ501.rOutPosition := FbMpbus_8.rOutPosition;
STLV80_360.STLV80_A_360_7C201_SQ501.rOutAirVolume_perc := FbMpbus_8.rOutAirVolume_perc;
STLV80_360.STLV80_A_360_7C201_SQ501.rOutAirVolume_m3h := FbMpbus_8.rOutAirVolume_m3_h;
STLV80_360.STLV80_A_360_7C201_SQ501.wSensorValue := FbMpbus_8.wSensorValue;
STLV80_360.STLV80_A_360_7C201_SQ501.rVmin := FbMpbus_8.rVmin;
STLV80_360.STLV80_A_360_7C201_SQ501.rVmax := FbMpbus_8.rVmax;
STLV80_360.STLV80_A_360_7C201_SQ501.xControlRangeIncreased := FbMpbus_8.xControlRangeIncreased;
STLV80_360.STLV80_A_360_7C201_SQ501.xMecanicalOverload := FbMpbus_8.xMecanicalOverload;
STLV80_360.STLV80_A_360_7C201_SQ501.xActuatorHunting := FbMpbus_8.xActuatorHunting;
STLV80_360.STLV80_A_360_7C201_SQ501.xSensorError := FbMpbus_8.xSensorError;
END_PROGRAM

PROGRAM PRG_MP2
  VAR
    xSet : BOOL;  (* Felles *)
    xRead : BOOL;
    FbMpbusMaster_2 : FbMpbusMaster;  (* Master *)
    oStatus_M2 : WagoSysErrorBase.FbResult;
    sStatus_M2 : STRING;
    FbMpbus_1 : FbMpBusVav;  (* Linje 2. Adresse 1. VAV STLV80_A_360_6G201_SQ401 *)
    oStatus_1 : WagoSysErrorBase.FbResult;
    sStatus_1 : STRING;
    FbMpbus_2 : FbMpBusVav;  (* Linje 2. Adresse 2. VAV STLV80_A_360_6M201_SQ503 *)
    oStatus_2 : WagoSysErrorBase.FbResult;
    sStatus_2 : STRING;
    FbMpbus_3 : FbMpBusVav;  (* Linje 2. Adresse 3. VAV STLV80_A_360_6M201_SQ403 *)
    oStatus_3 : WagoSysErrorBase.FbResult;
    sStatus_3 : STRING;
    FbMpbus_4 : FbMpBusVav;  (* Linje 2. Adresse 4. VAV STLV80_A_360_6M201_SQ402 *)
    oStatus_4 : WagoSysErrorBase.FbResult;
    sStatus_4 : STRING;
    FbMpbus_5 : FbMpBusVav;  (* Linje 2. Adresse 5. VAV STLV80_A_360_6M201_SQ502 *)
    oStatus_5 : WagoSysErrorBase.FbResult;
    sStatus_5 : STRING;
    FbMpbus_6 : FbMpBusVav;  (* Linje 2. Adresse 6. VAV STLV80_A_360_6M201_SQ501 *)
    oStatus_6 : WagoSysErrorBase.FbResult;
    sStatus_6 : STRING;
    FbMpbus_7 : FbMpBusVav;  (* Linje 2. Adresse 7. VAV STLV80_A_360_6M201_SQ401 *)
    oStatus_7 : WagoSysErrorBase.FbResult;
    sStatus_7 : STRING;
  END_VAR

(* CFC diagram, written out as Structured Text *)
FbMpbusMaster_2(I_Port := IoConfig_Globals.MP_Bus_Master_1, bPortMpBus := 2);
oStatus_M2 := FbMpbusMaster_2.oStatus;
sStatus_M2 := FbMpbusMaster_2.sStatus;
(* STLV80_A_360_6G201_SQ401 *)
FbMpbus_1(xEnable := STLV80_360.STLV80_A_360_6G201_SQ401.xEnable, bPortMpBus := 2, bAddress := 1, tCycleTime := t#500ms, rAirVolume := STLV80_360.STLV80_A_360_6G201_SQ401.rAirVolume_SP, rMinAirVolume := 0, rMaxAirVolume := 100, xSet := xSet, xRead := xRead, bSensorType := 0, xManualOpen := STLV80_360.STLV80_A_360_6G201_SQ401.xManualOpen, xManualClose := STLV80_360.STLV80_A_360_6G201_SQ401.xManualClose);
oStatus_1 := FbMpbus_1.oStatus;
sStatus_1 := FbMpbus_1.sStatus;
STLV80_360.STLV80_A_360_6G201_SQ401.xReady := FbMpbus_1.xReady;
STLV80_360.STLV80_A_360_6G201_SQ401.rOutPosition := FbMpbus_1.rOutPosition;
STLV80_360.STLV80_A_360_6G201_SQ401.rOutAirVolume_perc := FbMpbus_1.rOutAirVolume_perc;
STLV80_360.STLV80_A_360_6G201_SQ401.rOutAirVolume_m3h := FbMpbus_1.rOutAirVolume_m3_h;
STLV80_360.STLV80_A_360_6G201_SQ401.wSensorValue := FbMpbus_1.wSensorValue;
STLV80_360.STLV80_A_360_6G201_SQ401.rVmin := FbMpbus_1.rVmin;
STLV80_360.STLV80_A_360_6G201_SQ401.rVmax := FbMpbus_1.rVmax;
STLV80_360.STLV80_A_360_6G201_SQ401.xControlRangeIncreased := FbMpbus_1.xControlRangeIncreased;
STLV80_360.STLV80_A_360_6G201_SQ401.xMecanicalOverload := FbMpbus_1.xMecanicalOverload;
STLV80_360.STLV80_A_360_6G201_SQ401.xActuatorHunting := FbMpbus_1.xActuatorHunting;
STLV80_360.STLV80_A_360_6G201_SQ401.xSensorError := FbMpbus_1.xSensorError;
(* STLV80_A_360_6M201_SQ503 *)
FbMpbus_2(xEnable := STLV80_360.STLV80_A_360_6M201_SQ503.xEnable, bPortMpBus := 2, bAddress := 2, tCycleTime := t#500ms, rAirVolume := STLV80_360.STLV80_A_360_6M201_SQ503.rAirVolume_SP, rMinAirVolume := 0, rMaxAirVolume := 100, xSet := xSet, xRead := xRead, bSensorType := 0, xManualOpen := STLV80_360.STLV80_A_360_6M201_SQ503.xManualOpen, xManualClose := STLV80_360.STLV80_A_360_6M201_SQ503.xManualClose);
oStatus_2 := FbMpbus_2.oStatus;
sStatus_2 := FbMpbus_2.sStatus;
STLV80_360.STLV80_A_360_6M201_SQ503.xReady := FbMpbus_2.xReady;
STLV80_360.STLV80_A_360_6M201_SQ503.rOutPosition := FbMpbus_2.rOutPosition;
STLV80_360.STLV80_A_360_6M201_SQ503.rOutAirVolume_perc := FbMpbus_2.rOutAirVolume_perc;
STLV80_360.STLV80_A_360_6M201_SQ503.rOutAirVolume_m3h := FbMpbus_2.rOutAirVolume_m3_h;
STLV80_360.STLV80_A_360_6M201_SQ503.wSensorValue := FbMpbus_2.wSensorValue;
STLV80_360.STLV80_A_360_6M201_SQ503.rVmin := FbMpbus_2.rVmin;
STLV80_360.STLV80_A_360_6M201_SQ503.rVmax := FbMpbus_2.rVmax;
STLV80_360.STLV80_A_360_6M201_SQ503.xControlRangeIncreased := FbMpbus_2.xControlRangeIncreased;
STLV80_360.STLV80_A_360_6M201_SQ503.xMecanicalOverload := FbMpbus_2.xMecanicalOverload;
STLV80_360.STLV80_A_360_6M201_SQ503.xActuatorHunting := FbMpbus_2.xActuatorHunting;
STLV80_360.STLV80_A_360_6M201_SQ503.xSensorError := FbMpbus_2.xSensorError;
(* STLV80_A_360_6M201_SQ403 *)
FbMpbus_3(xEnable := STLV80_360.STLV80_A_360_6M201_SQ403.xEnable, bPortMpBus := 2, bAddress := 3, tCycleTime := t#500ms, rAirVolume := STLV80_360.STLV80_A_360_6M201_SQ403.rAirVolume_SP, rMinAirVolume := 0, rMaxAirVolume := 100, xSet := xSet, xRead := xRead, bSensorType := 0, xManualOpen := STLV80_360.STLV80_A_360_6M201_SQ403.xManualOpen, xManualClose := STLV80_360.STLV80_A_360_6M201_SQ403.xManualClose);
oStatus_3 := FbMpbus_3.oStatus;
sStatus_3 := FbMpbus_3.sStatus;
STLV80_360.STLV80_A_360_6M201_SQ403.xReady := FbMpbus_3.xReady;
STLV80_360.STLV80_A_360_6M201_SQ403.rOutPosition := FbMpbus_3.rOutPosition;
STLV80_360.STLV80_A_360_6M201_SQ403.rOutAirVolume_perc := FbMpbus_3.rOutAirVolume_perc;
STLV80_360.STLV80_A_360_6M201_SQ403.rOutAirVolume_m3h := FbMpbus_3.rOutAirVolume_m3_h;
STLV80_360.STLV80_A_360_6M201_SQ403.wSensorValue := FbMpbus_3.wSensorValue;
STLV80_360.STLV80_A_360_6M201_SQ403.rVmin := FbMpbus_3.rVmin;
STLV80_360.STLV80_A_360_6M201_SQ403.rVmax := FbMpbus_3.rVmax;
STLV80_360.STLV80_A_360_6M201_SQ403.xControlRangeIncreased := FbMpbus_3.xControlRangeIncreased;
STLV80_360.STLV80_A_360_6M201_SQ403.xMecanicalOverload := FbMpbus_3.xMecanicalOverload;
STLV80_360.STLV80_A_360_6M201_SQ403.xActuatorHunting := FbMpbus_3.xActuatorHunting;
STLV80_360.STLV80_A_360_6M201_SQ403.xSensorError := FbMpbus_3.xSensorError;
(* STLV80_A_360_6M201_SQ402 *)
FbMpbus_4(xEnable := STLV80_360.STLV80_A_360_6M201_SQ402.xEnable, bPortMpBus := 2, bAddress := 4, tCycleTime := t#500ms, rAirVolume := STLV80_360.STLV80_A_360_6M201_SQ402.rAirVolume_SP, rMinAirVolume := 0, rMaxAirVolume := 100, xSet := xSet, xRead := xRead, bSensorType := 0, xManualOpen := STLV80_360.STLV80_A_360_6M201_SQ402.xManualOpen, xManualClose := STLV80_360.STLV80_A_360_6M201_SQ402.xManualClose);
oStatus_4 := FbMpbus_4.oStatus;
sStatus_4 := FbMpbus_4.sStatus;
STLV80_360.STLV80_A_360_6M201_SQ402.xReady := FbMpbus_4.xReady;
STLV80_360.STLV80_A_360_6M201_SQ402.rOutPosition := FbMpbus_4.rOutPosition;
STLV80_360.STLV80_A_360_6M201_SQ402.rOutAirVolume_perc := FbMpbus_4.rOutAirVolume_perc;
STLV80_360.STLV80_A_360_6M201_SQ402.rOutAirVolume_m3h := FbMpbus_4.rOutAirVolume_m3_h;
STLV80_360.STLV80_A_360_6M201_SQ402.wSensorValue := FbMpbus_4.wSensorValue;
STLV80_360.STLV80_A_360_6M201_SQ402.rVmin := FbMpbus_4.rVmin;
STLV80_360.STLV80_A_360_6M201_SQ402.rVmax := FbMpbus_4.rVmax;
STLV80_360.STLV80_A_360_6M201_SQ402.xControlRangeIncreased := FbMpbus_4.xControlRangeIncreased;
STLV80_360.STLV80_A_360_6M201_SQ402.xMecanicalOverload := FbMpbus_4.xMecanicalOverload;
STLV80_360.STLV80_A_360_6M201_SQ402.xActuatorHunting := FbMpbus_4.xActuatorHunting;
STLV80_360.STLV80_A_360_6M201_SQ402.xSensorError := FbMpbus_4.xSensorError;
(* STLV80_A_360_6M201_SQ502 *)
FbMpbus_5(xEnable := STLV80_360.STLV80_A_360_6M201_SQ502.xEnable, bPortMpBus := 2, bAddress := 5, tCycleTime := t#500ms, rAirVolume := STLV80_360.STLV80_A_360_6M201_SQ502.rAirVolume_SP, rMinAirVolume := 0, rMaxAirVolume := 100, xSet := xSet, xRead := xRead, bSensorType := 0, xManualOpen := STLV80_360.STLV80_A_360_6M201_SQ502.xManualOpen, xManualClose := STLV80_360.STLV80_A_360_6M201_SQ502.xManualClose);
oStatus_5 := FbMpbus_5.oStatus;
sStatus_5 := FbMpbus_5.sStatus;
STLV80_360.STLV80_A_360_6M201_SQ502.xReady := FbMpbus_5.xReady;
STLV80_360.STLV80_A_360_6M201_SQ502.rOutPosition := FbMpbus_5.rOutPosition;
STLV80_360.STLV80_A_360_6M201_SQ502.rOutAirVolume_perc := FbMpbus_5.rOutAirVolume_perc;
STLV80_360.STLV80_A_360_6M201_SQ502.rOutAirVolume_m3h := FbMpbus_5.rOutAirVolume_m3_h;
STLV80_360.STLV80_A_360_6M201_SQ502.wSensorValue := FbMpbus_5.wSensorValue;
STLV80_360.STLV80_A_360_6M201_SQ502.rVmin := FbMpbus_5.rVmin;
STLV80_360.STLV80_A_360_6M201_SQ502.rVmax := FbMpbus_5.rVmax;
STLV80_360.STLV80_A_360_6M201_SQ502.xControlRangeIncreased := FbMpbus_5.xControlRangeIncreased;
STLV80_360.STLV80_A_360_6M201_SQ502.xMecanicalOverload := FbMpbus_5.xMecanicalOverload;
STLV80_360.STLV80_A_360_6M201_SQ502.xActuatorHunting := FbMpbus_5.xActuatorHunting;
STLV80_360.STLV80_A_360_6M201_SQ502.xSensorError := FbMpbus_5.xSensorError;
(* STLV80_A_360_6M201_SQ501 *)
FbMpbus_6(xEnable := STLV80_360.STLV80_A_360_6M201_SQ501.xEnable, bPortMpBus := 2, bAddress := 6, tCycleTime := t#500ms, rAirVolume := STLV80_360.STLV80_A_360_6M201_SQ501.rAirVolume_SP, rMinAirVolume := 0, rMaxAirVolume := 100, xSet := xSet, xRead := xRead, bSensorType := 0, xManualOpen := STLV80_360.STLV80_A_360_6M201_SQ501.xManualOpen, xManualClose := STLV80_360.STLV80_A_360_6M201_SQ501.xManualClose);
oStatus_6 := FbMpbus_6.oStatus;
sStatus_6 := FbMpbus_6.sStatus;
STLV80_360.STLV80_A_360_6M201_SQ501.xReady := FbMpbus_6.xReady;
STLV80_360.STLV80_A_360_6M201_SQ501.rOutPosition := FbMpbus_6.rOutPosition;
STLV80_360.STLV80_A_360_6M201_SQ501.rOutAirVolume_perc := FbMpbus_6.rOutAirVolume_perc;
STLV80_360.STLV80_A_360_6M201_SQ501.rOutAirVolume_m3h := FbMpbus_6.rOutAirVolume_m3_h;
STLV80_360.STLV80_A_360_6M201_SQ501.wSensorValue := FbMpbus_6.wSensorValue;
STLV80_360.STLV80_A_360_6M201_SQ501.rVmin := FbMpbus_6.rVmin;
STLV80_360.STLV80_A_360_6M201_SQ501.rVmax := FbMpbus_6.rVmax;
STLV80_360.STLV80_A_360_6M201_SQ501.xControlRangeIncreased := FbMpbus_6.xControlRangeIncreased;
STLV80_360.STLV80_A_360_6M201_SQ501.xMecanicalOverload := FbMpbus_6.xMecanicalOverload;
STLV80_360.STLV80_A_360_6M201_SQ501.xActuatorHunting := FbMpbus_6.xActuatorHunting;
STLV80_360.STLV80_A_360_6M201_SQ501.xSensorError := FbMpbus_6.xSensorError;
(* STLV80_A_360_6M201_SQ401 *)
FbMpbus_7(xEnable := STLV80_360.STLV80_A_360_6M201_SQ401.xEnable, bPortMpBus := 2, bAddress := 7, tCycleTime := t#500ms, rAirVolume := STLV80_360.STLV80_A_360_6M201_SQ401.rAirVolume_SP, rMinAirVolume := 0, rMaxAirVolume := 100, xSet := xSet, xRead := xRead, bSensorType := 0, xManualOpen := STLV80_360.STLV80_A_360_6M201_SQ401.xManualOpen, xManualClose := STLV80_360.STLV80_A_360_6M201_SQ401.xManualClose);
oStatus_7 := FbMpbus_7.oStatus;
sStatus_7 := FbMpbus_7.sStatus;
STLV80_360.STLV80_A_360_6M201_SQ401.xReady := FbMpbus_7.xReady;
STLV80_360.STLV80_A_360_6M201_SQ401.rOutPosition := FbMpbus_7.rOutPosition;
STLV80_360.STLV80_A_360_6M201_SQ401.rOutAirVolume_perc := FbMpbus_7.rOutAirVolume_perc;
STLV80_360.STLV80_A_360_6M201_SQ401.rOutAirVolume_m3h := FbMpbus_7.rOutAirVolume_m3_h;
STLV80_360.STLV80_A_360_6M201_SQ401.wSensorValue := FbMpbus_7.wSensorValue;
STLV80_360.STLV80_A_360_6M201_SQ401.rVmin := FbMpbus_7.rVmin;
STLV80_360.STLV80_A_360_6M201_SQ401.rVmax := FbMpbus_7.rVmax;
STLV80_360.STLV80_A_360_6M201_SQ401.xControlRangeIncreased := FbMpbus_7.xControlRangeIncreased;
STLV80_360.STLV80_A_360_6M201_SQ401.xMecanicalOverload := FbMpbus_7.xMecanicalOverload;
STLV80_360.STLV80_A_360_6M201_SQ401.xActuatorHunting := FbMpbus_7.xActuatorHunting;
STLV80_360.STLV80_A_360_6M201_SQ401.xSensorError := FbMpbus_7.xSensorError;
END_PROGRAM

PROGRAM PRG_MP3
  VAR
    xSet : BOOL;  (* Felles *)
    xRead : BOOL;
    FbMpbusMaster_3 : FbMpbusMaster;  (* Master *)
    oStatus_M3 : WagoSysErrorBase.FbResult;
    sStatus_M3 : STRING;
    FbMpbus_1 : FbMpBusVav;  (* Linje 3. Adresse 1. VAV STLV80_A_360_7O201_SQ401 *)
    oStatus_1 : WagoSysErrorBase.FbResult;
    sStatus_1 : STRING;
    FbMpbus_2 : FbMpBusVav;  (* Linje 3. Adresse 2. VAV STLV80_A_360_7O201_SQ501 *)
    oStatus_2 : WagoSysErrorBase.FbResult;
    sStatus_2 : STRING;
  END_VAR

(* CFC diagram, written out as Structured Text *)
FbMpbusMaster_3(I_Port := IoConfig_Globals.MP_Bus_Master_2, bPortMpBus := 3);
oStatus_M3 := FbMpbusMaster_3.oStatus;
sStatus_M3 := FbMpbusMaster_3.sStatus;
(* STLV80_A_360_7O201_SQ401 *)
FbMpbus_1(xEnable := STLV80_360.STLV80_A_360_7O201_SQ401.xEnable, bPortMpBus := 3, bAddress := 1, tCycleTime := t#500ms, rAirVolume := STLV80_360.STLV80_A_360_7O201_SQ401.rAirVolume_SP, rMinAirVolume := 0, rMaxAirVolume := 100, xSet := xSet, xRead := xRead, bSensorType := 0, xManualOpen := STLV80_360.STLV80_A_360_7O201_SQ401.xManualOpen, xManualClose := STLV80_360.STLV80_A_360_7O201_SQ401.xManualClose);
oStatus_1 := FbMpbus_1.oStatus;
sStatus_1 := FbMpbus_1.sStatus;
STLV80_360.STLV80_A_360_7O201_SQ401.xReady := FbMpbus_1.xReady;
STLV80_360.STLV80_A_360_7O201_SQ401.rOutPosition := FbMpbus_1.rOutPosition;
STLV80_360.STLV80_A_360_7O201_SQ401.rOutAirVolume_perc := FbMpbus_1.rOutAirVolume_perc;
STLV80_360.STLV80_A_360_7O201_SQ401.rOutAirVolume_m3h := FbMpbus_1.rOutAirVolume_m3_h;
STLV80_360.STLV80_A_360_7O201_SQ401.wSensorValue := FbMpbus_1.wSensorValue;
STLV80_360.STLV80_A_360_7O201_SQ401.rVmin := FbMpbus_1.rVmin;
STLV80_360.STLV80_A_360_7O201_SQ401.rVmax := FbMpbus_1.rVmax;
STLV80_360.STLV80_A_360_7O201_SQ401.xControlRangeIncreased := FbMpbus_1.xControlRangeIncreased;
STLV80_360.STLV80_A_360_7O201_SQ401.xMecanicalOverload := FbMpbus_1.xMecanicalOverload;
STLV80_360.STLV80_A_360_7O201_SQ401.xActuatorHunting := FbMpbus_1.xActuatorHunting;
STLV80_360.STLV80_A_360_7O201_SQ401.xSensorError := FbMpbus_1.xSensorError;
(* STLV80_A_360_7O201_SQ501 *)
FbMpbus_2(xEnable := STLV80_360.STLV80_A_360_7O201_SQ501.xEnable, bPortMpBus := 3, bAddress := 2, tCycleTime := t#500ms, rAirVolume := STLV80_360.STLV80_A_360_7O201_SQ501.rAirVolume_SP, rMinAirVolume := 0, rMaxAirVolume := 100, xSet := xSet, xRead := xRead, bSensorType := 0, xManualOpen := STLV80_360.STLV80_A_360_7O201_SQ501.xManualOpen, xManualClose := STLV80_360.STLV80_A_360_7O201_SQ501.xManualClose);
oStatus_2 := FbMpbus_2.oStatus;
sStatus_2 := FbMpbus_2.sStatus;
STLV80_360.STLV80_A_360_7O201_SQ501.xReady := FbMpbus_2.xReady;
STLV80_360.STLV80_A_360_7O201_SQ501.rOutPosition := FbMpbus_2.rOutPosition;
STLV80_360.STLV80_A_360_7O201_SQ501.rOutAirVolume_perc := FbMpbus_2.rOutAirVolume_perc;
STLV80_360.STLV80_A_360_7O201_SQ501.rOutAirVolume_m3h := FbMpbus_2.rOutAirVolume_m3_h;
STLV80_360.STLV80_A_360_7O201_SQ501.wSensorValue := FbMpbus_2.wSensorValue;
STLV80_360.STLV80_A_360_7O201_SQ501.rVmin := FbMpbus_2.rVmin;
STLV80_360.STLV80_A_360_7O201_SQ501.rVmax := FbMpbus_2.rVmax;
STLV80_360.STLV80_A_360_7O201_SQ501.xControlRangeIncreased := FbMpbus_2.xControlRangeIncreased;
STLV80_360.STLV80_A_360_7O201_SQ501.xMecanicalOverload := FbMpbus_2.xMecanicalOverload;
STLV80_360.STLV80_A_360_7O201_SQ501.xActuatorHunting := FbMpbus_2.xActuatorHunting;
STLV80_360.STLV80_A_360_7O201_SQ501.xSensorError := FbMpbus_2.xSensorError;
END_PROGRAM
